TEXTLIST GLP_Status
  0 = 'Off'
  1 = 'On'
   = ''
END_TEXTLIST

(* stored: Version 1.1.0.1, ProductVersion 3.1.4024.12
   TextList GLP_Status: Id {33065706-f2c8-4784-bfd9-85fbb99f7071} *)
